% RSLogix 500 project TASK_BAK019.RSS, saved by version 8.10.00.18 %
PROJECT "UNTITLED"    % processor: MicroLogix 1200 %

PROGRAM FILES
  LAD 2   8 rungs

DATA FILES
  O0 OUTPUT  4 elements
  I1 INPUT  4 elements
  S2 STATUS  66 elements
  B3 BINARY  1 elements
  T4 TIMER  2 elements
  C5 COUNTER  1 elements
  R6 CONTROL  1 elements
  N7 INTEGER  1 elements

LADDER 2
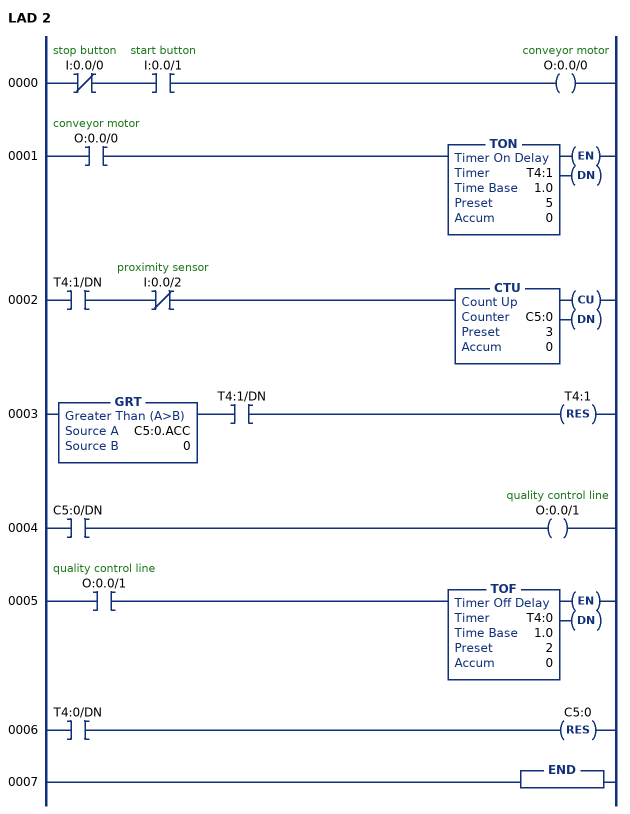
% Rung: 0 %
SOR XIO I:0.0/0 XIC I:0.0/1 OTE O:0.0/0 EOR
%   I:0.0/0  "stop button" %
%   I:0.0/1  "start button" %
%   O:0.0/0  "conveyor motor" %
% Rung: 1 %
SOR XIC O:0.0/0 TON T4:1 1.0 5 0 EOR
%   O:0.0/0  "conveyor motor" %
% Rung: 2 %
SOR XIC T4:1/DN XIO I:0.0/2 CTU C5:0 3 0 EOR
%   I:0.0/2  "proximity sensor" %
% Rung: 3 %
SOR GRT C5:0.ACC 0 XIC T4:1/DN RES T4:1 EOR
% Rung: 4 %
SOR XIC C5:0/DN OTE O:0.0/1 EOR
%   O:0.0/1  "quality control line" %
% Rung: 5 %
SOR XIC O:0.0/1 TOF T4:0 1.0 2 0 EOR
%   O:0.0/1  "quality control line" %
% Rung: 6 %
SOR XIC T4:0/DN RES C5:0 EOR
% Rung: 7 %
SOR END EOR

OTHER DOCUMENTED ADDRESSES
  O:0.0/2  "proximity sensor"

DATA TABLE (non-zero values as saved)
DATA T4
% .PRE .ACC %
% T4:0 % 2 0
% T4:1 % 5 0
DATA C5
% .PRE .ACC %
% C5:0 % 3 0
